INTERFACE I_FREQ_GEN EXTENDS I_GENERAL_OBJECT

METHOD M_SetFrequence : bool
VAR_INPUT
	iFreqence: INT;
END_VAR
END_METHOD

PROPERTY P_FTrig : BOOL
GET
END_GET
END_PROPERTY

PROPERTY P_RTrig : BOOL
GET
END_GET
END_PROPERTY

PROPERTY P_State : BOOL
GET
END_GET
END_PROPERTY

END_INTERFACE

(* stored: Version 1.1.0.1, ProductVersion 3.1.4024.12
   Itf I_FREQ_GEN: Id {5577f50f-75cb-4667-9173-3b42f861a128}
   Method M_SetFrequence: Id {53805b9a-c123-49cf-b720-9951ac3f826f}
   Property P_FTrig: Id {783a0e9f-4e64-47ad-b880-d7345c7c7907}
   Get Get: Id {7e196938-0097-4b2c-8b89-293156a582d6}
   Property P_RTrig: Id {84eb4340-1e90-47bc-a4a9-10fac0fad250}
   Get Get: Id {5d62675f-dc16-466f-bc28-c7decf647d6c}
   Property P_State: Id {dad35a53-8995-46d6-be28-36d5be4a8120}
   Get Get: Id {25647814-807e-495c-bc76-eeed59e75c75} *)
